{attribute 'linkalways'} 
{attribute 'no_explicit_call' := 'This FB is a CLASS and must be accessed using methods or properties'}
{attribute 'enable_dynamic_creation'}
FUNCTION_BLOCK FINAL XOR_UINT EXTENDS Node
VAR
	in1 : _UINT(0);
	in2 : _UINT(0);
	out : _UINT(0);
END_VAR

METHOD PUBLIC Clone : I_Node
VAR
	pNode : POINTER TO XOR_UINT;
END_VAR
pNode := __NEW(XOR_UINT);
Clone := pNode^;
END_METHOD

METHOD FB_init : BOOL
VAR_INPUT
	bInitRetains : BOOL; // if TRUE, the retain variables are initialized (warm start / cold start)
	bInCopyCode : BOOL;  // if TRUE, the instance afterwards gets moved into the copy code (online change)
END_VAR
AddInput('in1',THIS^.in1);
AddInput('in2',THIS^.in2);
AddOutput('out', THIS^.out);
END_METHOD

METHOD PROTECTED OnExecute
VAR
END_VAR
out.Value := in1.Value XOR in2.Value;
END_METHOD

END_FUNCTION_BLOCK

(* stored: Version 1.1.0.1, ProductVersion 3.1.4024.15
   POU XOR_UINT: Id {d2e19beb-eb72-4184-b3b9-664c113d7e95}, SpecialFunc None
   Folder Constructor: Id {91fe2e88-4c56-4224-bda2-bb819d7aa3bd}
   Method Clone: Id {13236a8f-40ee-4a28-ad5b-6f8e53ec0287}
   Method FB_init: Id {62d77378-4072-4b93-9b21-4dc6ae923a45}
   Method OnExecute: Id {72c80fc7-c505-4c7e-a4b7-9cee1fd08c48} *)
